(* PLC project Tc3_EventLogger.FB_RequestEventText Demo, tc3-libraries-kb TwinCAT 3.1 *)
(* stored: creationDateTime 2026-05-11T01:00:00, modificationDateTime 2026-05-11T01:00:00 *)

PROGRAM P_Demo_FB_RequestEventText
  VAR
    fbFB_RequestEventText : FB_RequestEventText;  (* Tc3_EventLogger.FB_RequestEventText 实例 *)
    arg_sResult : REFERENCE TO STRING;  (* VAR_INPUT sResult *)
    arg_nResult : UDINT;  (* VAR_INPUT nResult *)
    arg_eventClass : GUID;  (* VAR_INPUT eventClass *)
    arg_nEventId : UDINT;  (* VAR_INPUT nEventId *)
    arg_nLangId : DINT;  (* VAR_INPUT nLangId *)
    arg_ipArgs : I_TcArguments;  (* VAR_INPUT ipArgs *)
    arg_ipRemoteLogger : I_TcRemoteEventLogger;  (* VAR_INPUT ipRemoteLogger *)
  END_VAR

            // ============================================================
// Tc3_EventLogger.FB_RequestEventText 演示程序（FB 实例）
// ============================================================
// 验证步骤：
//   1. 引用 Tc3_EventLogger（及依赖类型所在库 Tc2_System 等）
//   2. 编译 + 登录
//   3. 按 doc.md 给 arg_* 赋值
//   4. 在线监视 out_* / io_* 输出
// ============================================================

fbFB_RequestEventText(
    sResult := arg_sResult,
    nResult := arg_nResult,
    eventClass := arg_eventClass,
    nEventId := arg_nEventId,
    nLangId := arg_nLangId,
    ipArgs := arg_ipArgs,
    ipRemoteLogger := arg_ipRemoteLogger
);

          
END_PROGRAM
